{region '#Template'}
	{attribute 'Version' := '5.1.0.0'}
	{attribute 'Tags' := '"LCID": "1031", "Text": "RA, HC, Building, Setpoint"'}
	{attribute 'Tags' := '"LCID": "1033", "Text": "RA, HC, Building, Setpoint"'}
	{attribute 'Using' := '"Type": "Template", "URI": "Site"'}
	{attribute 'Description' := '"LCID": "1031", "Text": "Gebäude Temperatursollwerte Raum"'}
	{attribute 'Description' := '"LCID": "1033", "Text": "Building temperature-setpoints room"'}
{endregion}
FUNCTION_BLOCK FB_BA_BuildingSpRmT EXTENDS FB_BA_View
VAR_INPUT CONSTANT    	
	SumCpsn					: FB_BA_Scale_02;
	WinCpsn					: FB_BA_Scale_02;                                  
	PrtcHtg					: FB_BA_AV_Op;           
	EcoHtg					: FB_BA_AV_Op;          
	PreCmfHtg				: FB_BA_AV_Op;          
	CmfHtg					: FB_BA_AV_Op;            
	PrtcCol					: FB_BA_AV_Op;          
	EcoCol					: FB_BA_AV_Op;        
	PreCmfCol				: FB_BA_AV_Op;         
	CmfCol					: FB_BA_AV_Op;            
	ShiftHtg				: FB_BA_AV_Op;             
	ShiftCol				: FB_BA_AV_Op;        
END_VAR                     
                            
VAR	                        
	SpRmT					: FB_BA_SpRmT;
END_VAR

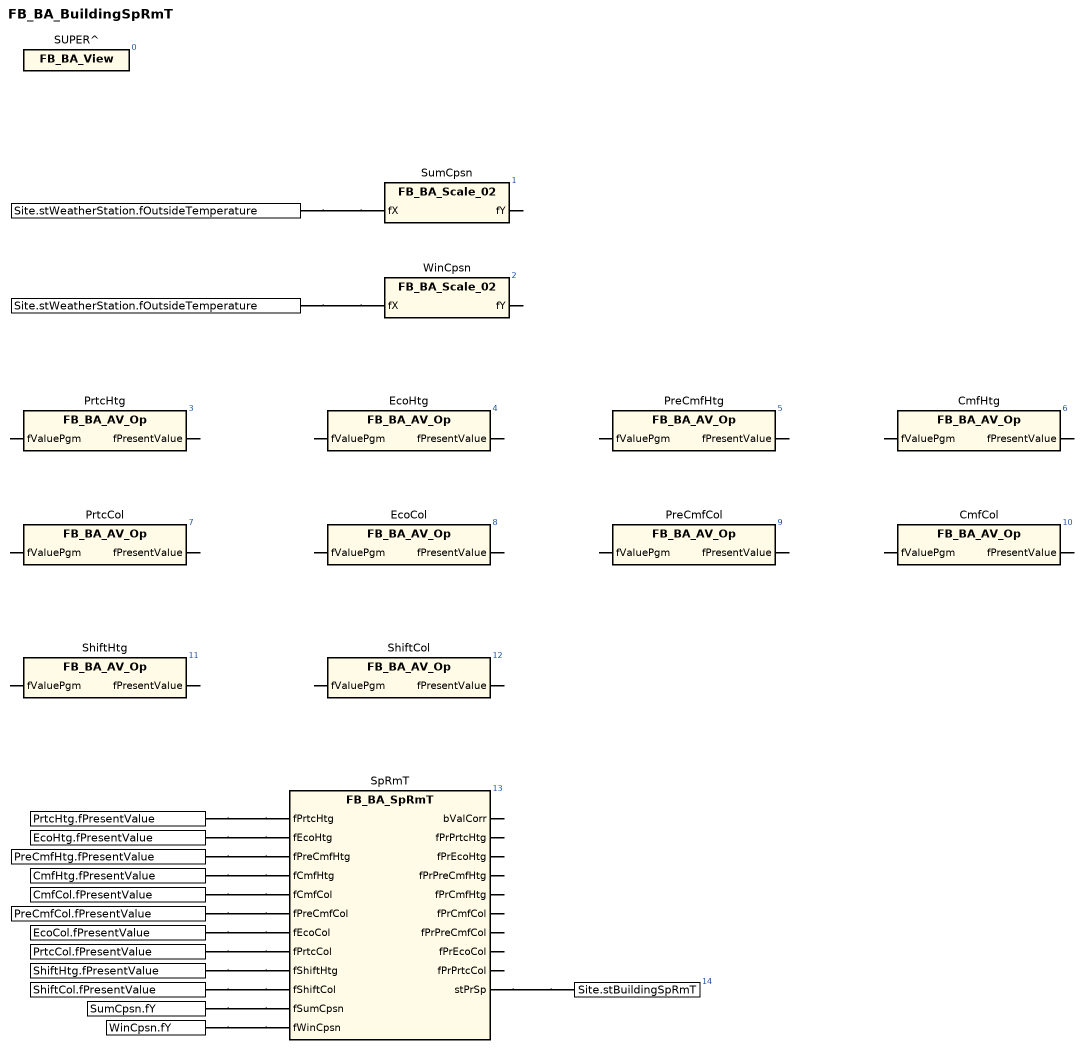
SUPER^(); // FB_BA_View
SumCpsn(fX := Site.stWeatherStation.fOutsideTemperature); // FB_BA_Scale_02
WinCpsn(fX := Site.stWeatherStation.fOutsideTemperature); // FB_BA_Scale_02
PrtcHtg(); // FB_BA_AV_Op
EcoHtg(); // FB_BA_AV_Op
PreCmfHtg(); // FB_BA_AV_Op
CmfHtg(); // FB_BA_AV_Op
PrtcCol(); // FB_BA_AV_Op
EcoCol(); // FB_BA_AV_Op
PreCmfCol(); // FB_BA_AV_Op
CmfCol(); // FB_BA_AV_Op
ShiftHtg(); // FB_BA_AV_Op
ShiftCol(); // FB_BA_AV_Op
SpRmT(
    fPrtcHtg := PrtcHtg.fPresentValue,
    fEcoHtg := EcoHtg.fPresentValue,
    fPreCmfHtg := PreCmfHtg.fPresentValue,
    fCmfHtg := CmfHtg.fPresentValue,
    fCmfCol := CmfCol.fPresentValue,
    fPreCmfCol := PreCmfCol.fPresentValue,
    fEcoCol := EcoCol.fPresentValue,
    fPrtcCol := PrtcCol.fPresentValue,
    fShiftHtg := ShiftHtg.fPresentValue,
    fShiftCol := ShiftCol.fPresentValue,
    fSumCpsn := SumCpsn.fY,
    fWinCpsn := WinCpsn.fY); // FB_BA_SpRmT
Site.stBuildingSpRmT := SpRmT.stPrSp;

METHOD FB_init : BOOL
VAR_INPUT
	bInitRetains : BOOL; // if TRUE; the retain variables are initialized (warm start / cold start)
	bInCopyCode : BOOL;  // if TRUE; the instance afterwards gets moved into the copy code (online change)
END_VAR
SumCpsn.iParent				:= THIS^;	
SumCpsn.iLabel				:= LblCtl_SummerCompensation;						 
SumCpsn.eDPADMode			:= E_BA_DPADMode.eIncludeDescription;
SumCpsn.X1.fValueRm			:= 24.0;
SumCpsn.X2.fValueRm			:= 30.0;
SumCpsn.Y1.fValueRm			:= 0.0;
SumCpsn.Y2.fValueRm			:= 5.0;
SumCpsn.YMin.fValueRm		:= 0.0;
SumCpsn.YMax.fValueRm		:= 5.0;
                        	
WinCpsn.iParent				:= THIS^;	
WinCpsn.iLabel				:= LblCtl_WinterCompensation;
WinCpsn.eDPADMode			:= E_BA_DPADMode.eIncludeDescription;	
WinCpsn.X1.fValueRm			:= 10.0;
WinCpsn.X2.fValueRm			:= 0.0;
WinCpsn.Y1.fValueRm			:= 0.0;
WinCpsn.Y2.fValueRm			:= 2.0;
WinCpsn.YMin.fValueRm		:= 0.0;
WinCpsn.YMax.fValueRm		:= 2.0;
                                   
PrtcHtg.iParent				:= THIS^;
PrtcHtg.iLabel				:= LblFun_SetpointProtectionHeating;	
PrtcHtg.fValueRm			:= 12.0;
PrtcHtg.eUnit				:= E_BA_Unit.eTemperature_DegreesCelsius;

EcoHtg.iParent				:= THIS^;
EcoHtg.iLabel				:= LblFun_SetpointEconomyHeating;
EcoHtg.fValueRm				:= 15.0;
EcoHtg.eUnit				:= E_BA_Unit.eTemperature_DegreesCelsius;	

PreCmfHtg.iParent			:= THIS^;
PreCmfHtg.iLabel			:= LblFun_SetpointPreComfortHeating;
PreCmfHtg.fValueRm			:= 19.0;
PreCmfHtg.eUnit				:= E_BA_Unit.eTemperature_DegreesCelsius;

CmfHtg.iParent				:= THIS^;
CmfHtg.iLabel				:= LblFun_SetpointComfortHeating;		
CmfHtg.fValueRm				:= 21.0;
CmfHtg.eUnit				:= E_BA_Unit.eTemperature_DegreesCelsius;

PrtcCol.iParent				:= THIS^;
PrtcCol.iLabel				:= LblFun_SetpointProtectionCooling;
PrtcCol.fValueRm			:= 40.0;
PrtcCol.eUnit				:= E_BA_Unit.eTemperature_DegreesCelsius;

EcoCol.iParent				:= THIS^;
EcoCol.iLabel				:= LblFun_SetpointEconomyCooling;
EcoCol.fValueRm				:= 35.0;
EcoCol.eUnit				:= E_BA_Unit.eTemperature_DegreesCelsius;

PreCmfCol.iParent			:= THIS^;
PreCmfCol.iLabel			:= LblFun_SetpointPreComfortCooling;
PreCmfCol.fValueRm			:= 28.0;
PreCmfCol.eUnit				:= E_BA_Unit.eTemperature_DegreesCelsius;

CmfCol.iParent				:= THIS^;
CmfCol.iLabel				:= LblFun_SetpointComfortCooling;
CmfCol.fValueRm				:= 24.0;
CmfCol.eUnit				:= E_BA_Unit.eTemperature_DegreesCelsius;

ShiftHtg.iParent			:= THIS^;
ShiftHtg.iLabel				:= LblCtl_SetpointShiftHeating;
ShiftHtg.fValueRm			:= 0.0;
ShiftHtg.eUnit				:= E_BA_Unit.eTemperature_DegreesKelvin;

ShiftCol.iParent			:= THIS^;
ShiftCol.iLabel				:= LblCtl_SetpointShiftCooling;
ShiftCol.fValueRm			:= 0.0;
ShiftCol.eUnit				:= E_BA_Unit.eTemperature_DegreesKelvin;
END_METHOD

END_FUNCTION_BLOCK

(* stored: Version 1.1.0.1, ProductVersion 3.1.4024.12
   POU FB_BA_BuildingSpRmT: Id {91727ead-fab9-4ac1-8561-03745ce29cf0}, SpecialFunc None
   Method FB_init: Id {5aef73d6-9ae4-41d6-bc7f-e950302d8535} *)
